{attribute 'pack_mode' := '2'}
TYPE ST_NCI_M_FUNC :
STRUCT
  FastMFuncMask   : ARRAY [1..5] OF DWORD;
  HskMFuncNo      : UINT;
  HskMFuncReq     : WORD;
  HFuncValue      : UDINT; 

  MFuncGranted    : UINT;
END_STRUCT
END_TYPE

(* stored: Version 1.1.0.1, ProductVersion 3.1.4024.12
   DUT ST_NCI_M_FUNC: Id {84efd054-6a78-06df-2985-5b753ea81a5d} *)
